PROGRAM INDEP
VAR
END_VAR

END_PROGRAM

(* stored: Version 1.1.0.1, ProductVersion 3.1.4022.18
   POU INDEP: Id {14ae7ba1-7509-475f-af40-69a58bd85d3b}, SpecialFunc None *)
